# EPICS autosave request: iocBoot/iocTestBusyAsyn/auto_settings.req
file testBusyAsyn_settings.req P=$(P)
